INTERFACE I_Notify EXTENDS I_Object

METHOD M_Notify
VAR_INPUT
	stEvent:		ST_Event;
END_VAR
END_METHOD

END_INTERFACE

(* stored: Version 1.1.0.1
   Itf I_Notify: Id {57d1f153-b955-0712-06ba-6b2be9fbd0f9}
   Method M_Notify: Id {d0a0ed14-7b79-0120-0441-d1a3d375e475} *)
